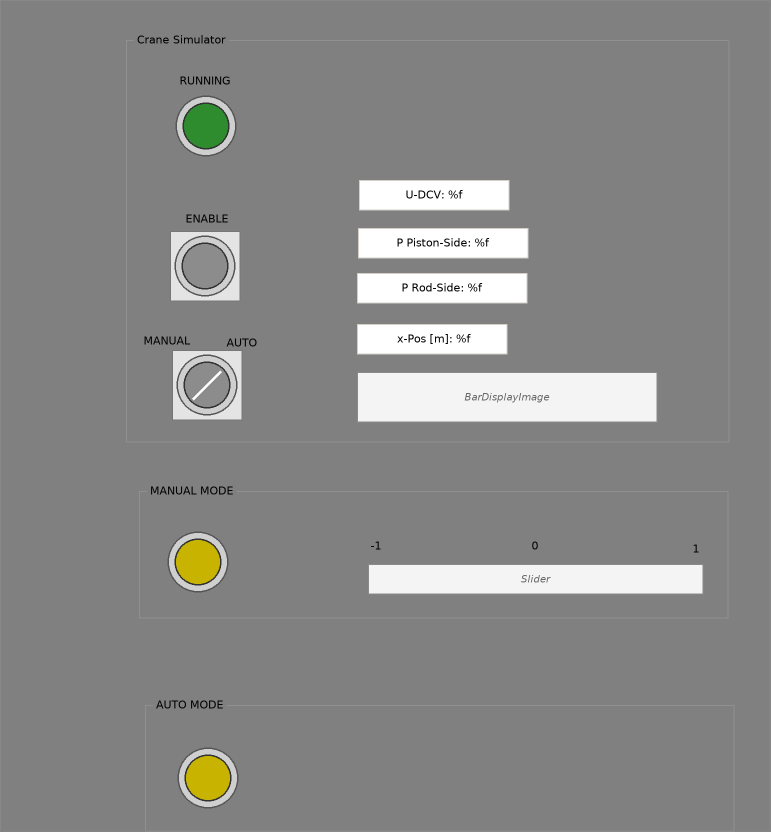
VISUALIZATION Visualization  // 771x832
    GroupBox (126,32 603x410), "Crane Simulator"
        Lamp1 (45,59 70x70), variable: P_Simulator.bSimulatorOn, style: Lamp-Lamp1-Green
        PushSwitch (44,199 70x70), variable: P_Simulator.bSimulatorOn, behaviour: TOGGLE, style: Switch-PushSwitch-Gray
        Textfield (233,148 150x30), "U-DCV: %f", text variable: P_Simulator.fUDCV
        Textfield (231,292 150x30), "x-Pos [m]: %f", text variable: P_Simulator.fCylPos
        Textfield (232,196 170x30), "P Piston-Side: %f", text variable: P_Simulator.fPpBar
        Textfield (231,241 170x30), "P Rod-Side: %f", text variable: P_Simulator.fPrBar
        BarDisplayImage (231,340 300x50), value: P_Simulator.fCylPos, style: BarDisplayImage-Gray, scale format: %.1f, scale 0..0.5
            p518627256: m
        Label (4,34 150x30), "RUNNING"
        Label (6,172 150x30), "ENABLE"
        RotarySwitch (46,318 70x70), variable: HMI.bAuto, behaviour: TOGGLE, style: Switch-RotarySwitch-Gray
        Label (41,296 150x30), "AUTO"
    Label (92,326 150x30), "MANUAL"
    GroupBox (139,483 589x135), "MANUAL MODE"
        Slider (229,81 335x30), variable: P_Simulator.fUDCV, scale -1..1
        Label (321,48 150x30), "0"
        Lamp1 (24,44 70x70), variable: HMI.bAuto, style: Lamp-Lamp1-Yellow
    Label (301,531 150x30), "-1"
    Label (621,534 150x30), "1"
    GroupBox (145,697 589x135), "AUTO MODE"
        Lamp1 (28,46 70x70), variable: NOT HMI.bAuto, style: Lamp-Lamp1-Yellow
END_VISUALIZATION

(* stored: Version 1.1.0.1, ProductVersion 3.1.4024.12
   Visu Visualization: Id {f1032fe3-236a-4d2f-8280-1a507172ce6c} *)
